Staubli VAL3: closeGripper.pgx

program closeGripper()
begin
  switchGripper=false
  taskKill("closeGripper")
end
